(* IEC 61131-3 sources: volt/packages/volt-lsp-iec/libraries/StringUtils/3.5.18.0, 27 files *)

(* ---- CHARTOUPPER.pou ---- *)
FUNCTION CHARTOUPPER : BYTE
VAR_INPUT
	BYCHAR : BYTE;
END_VAR
(* ASCII only: a..z become A..Z, every other byte is itself *)
IF BYCHAR >= 16#61 AND BYCHAR <= 16#7A THEN
	CHARTOUPPER := BYCHAR - 16#20;
ELSE
	CHARTOUPPER := BYCHAR;
END_IF
END_FUNCTION

(* ---- HELPISSAMEIGNORECASE.pou ---- *)
FUNCTION HELPISSAMEIGNORECASE : BOOL
VAR_INPUT
	BY1 : BYTE;
	BY2 : BYTE;
END_VAR
HELPISSAMEIGNORECASE := CHARTOUPPER(BY1) = CHARTOUPPER(BY2);
END_FUNCTION

(* ---- HELPSTRCMPENDA.pou ---- *)
FUNCTION HELPSTRCMPENDA : BOOL
VAR_INPUT
	PCOMPLETETEXT : CharBufferPtr;
	PSUBTEXT : CharBufferPtr;
	XIGNORECASE : BOOL;
END_VAR
VAR
	i : DINT;
	n : DINT;
	m : DINT;
END_VAR
(* does PCOMPLETETEXT end with PSUBTEXT (case folded when XIGNORECASE) *)
IF PCOMPLETETEXT = 0 OR PSUBTEXT = 0 THEN
	RETURN;
END_IF
n := STRLENA(PCOMPLETETEXT);
m := STRLENA(PSUBTEXT);
IF m > n THEN
	RETURN;
END_IF
FOR i := 0 TO m - 1 DO
	IF XIGNORECASE THEN
		IF NOT HELPISSAMEIGNORECASE(PCOMPLETETEXT[n - m + i], PSUBTEXT[i]) THEN
			RETURN;
		END_IF
	ELSIF PCOMPLETETEXT[n - m + i] <> PSUBTEXT[i] THEN
		RETURN;
	END_IF
END_FOR
HELPSTRCMPENDA := TRUE;
END_FUNCTION

(* ---- HELPSTRCMPSTARTA.pou ---- *)
FUNCTION HELPSTRCMPSTARTA : BOOL
VAR_INPUT
	PCOMPLETETEXT : CharBufferPtr;
	PSUBTEXT : CharBufferPtr;
	XIGNORECASE : BOOL;
END_VAR
VAR
	i : DINT;
END_VAR
(* does PCOMPLETETEXT begin with PSUBTEXT — every byte of it, in order (case folded when XIGNORECASE) *)
IF PCOMPLETETEXT = 0 OR PSUBTEXT = 0 THEN
	RETURN;
END_IF
WHILE PSUBTEXT[i] <> 0 DO
	IF PCOMPLETETEXT[i] = 0 THEN
		RETURN;
	END_IF
	IF XIGNORECASE THEN
		IF NOT HELPISSAMEIGNORECASE(PCOMPLETETEXT[i], PSUBTEXT[i]) THEN
			RETURN;
		END_IF
	ELSIF PCOMPLETETEXT[i] <> PSUBTEXT[i] THEN
		RETURN;
	END_IF
	i := i + 1;
END_WHILE
HELPSTRCMPSTARTA := TRUE;
END_FUNCTION

(* ---- ISSPACECHARACTER.pou ---- *)
FUNCTION ISSPACECHARACTER : BOOL
VAR_INPUT
	WCHARACTER : WORD;
END_VAR
(* a space, one of the control characters TAB, LF, VT, FF, CR, or the no-break space 16#A0 (recorded: lib_stu_chars).
   ponytail: the other Unicode spaces (16#2000.., 16#3000) are unasked — a fixture decides them *)
ISSPACECHARACTER := WCHARACTER = 16#20 OR (WCHARACTER >= 16#09 AND WCHARACTER <= 16#0D) OR WCHARACTER = 16#A0;
END_FUNCTION

(* ---- STRCASECMPA.pou ---- *)
FUNCTION STRCASECMPA : INT
VAR_INPUT
	PBYTE1 : POINTER TO BYTE;
	PBYTE2 : POINTER TO BYTE;
END_VAR
VAR
	i : DINT;
END_VAR
(* ignoring case (ASCII), how the first bytes that differ order: -1 when PBYTE1's is lower, 1 when higher, 0 when the
   strings are equal — the sign only (recorded: lib_stu_compare) *)
IF PBYTE1 = 0 OR PBYTE2 = 0 THEN
	RETURN;
END_IF
WHILE PBYTE1[i] <> 0 AND_THEN CHARTOUPPER(PBYTE1[i]) = CHARTOUPPER(PBYTE2[i]) DO
	i := i + 1;
END_WHILE
IF CHARTOUPPER(PBYTE1[i]) < CHARTOUPPER(PBYTE2[i]) THEN
	STRCASECMPA := -1;
ELSIF CHARTOUPPER(PBYTE1[i]) > CHARTOUPPER(PBYTE2[i]) THEN
	STRCASECMPA := 1;
END_IF
END_FUNCTION

(* ---- STRCASECMPENDA.pou ---- *)
FUNCTION STRCASECMPENDA : INT
VAR_INPUT
	PSTRING : CharBufferPtr;
	PSUFFIX : CharBufferPtr;
END_VAR
(* 0 when PSTRING ends with PSUFFIX, ignoring case — the answer a compare gives for equal — and -1 when it does not *)
IF HELPSTRCMPENDA(PSTRING, PSUFFIX, TRUE) THEN
	STRCASECMPENDA := 0;
ELSE
	STRCASECMPENDA := -1;
END_IF
END_FUNCTION

(* ---- STRCASECMPSTARTA.pou ---- *)
FUNCTION STRCASECMPSTARTA : INT
VAR_INPUT
	PSTRING : CharBufferPtr;
	PPREFIX : CharBufferPtr;
END_VAR
(* 0 when PSTRING begins with PPREFIX, ignoring case — the answer a compare gives for equal — and -1 when it does not *)
IF HELPSTRCMPSTARTA(PSTRING, PPREFIX, TRUE) THEN
	STRCASECMPSTARTA := 0;
ELSE
	STRCASECMPSTARTA := -1;
END_IF
END_FUNCTION

(* ---- STRCASECMPW.pou ---- *)
FUNCTION STRCASECMPW : INT
VAR_INPUT
	PWD1 : POINTER TO WORD;
	PWD2 : POINTER TO WORD;
END_VAR
VAR
	i : DINT;
END_VAR
(* ignoring case (ASCII), how the first words that differ order: -1 when PWD1's is lower, 1 when higher, 0 when the
   strings are equal — the sign only (recorded: lib_stu_compare) *)
IF PWD1 = 0 OR PWD2 = 0 THEN
	RETURN;
END_IF
WHILE PWD1[i] <> 0 AND_THEN WCHARTOUPPER(PWD1[i]) = WCHARTOUPPER(PWD2[i]) DO
	i := i + 1;
END_WHILE
IF WCHARTOUPPER(PWD1[i]) < WCHARTOUPPER(PWD2[i]) THEN
	STRCASECMPW := -1;
ELSIF WCHARTOUPPER(PWD1[i]) > WCHARTOUPPER(PWD2[i]) THEN
	STRCASECMPW := 1;
END_IF
END_FUNCTION

(* ---- STRCASEFINDA.pou ---- *)
FUNCTION STRCASEFINDA : INT
VAR_INPUT
	PST1 : POINTER TO STRING(255);
	PST2 : POINTER TO STRING(255);
	UISEARCHSTART : UINT;
END_VAR
VAR
	i : DINT;
	j : DINT;
	n1 : DINT;
	n2 : DINT;
END_VAR
(* where PST2 first occurs in PST1, ignoring case (ASCII), searching from UISEARCHSTART (counted from 1; 0 counts as 1)
   — the position counted from 1, or 0 when it does not occur. An empty PST2 occurs nowhere. *)
IF PST1 = 0 OR PST2 = 0 THEN
	RETURN;
END_IF
WHILE PST1^[n1] <> 0 DO
	n1 := n1 + 1;
END_WHILE
WHILE PST2^[n2] <> 0 DO
	n2 := n2 + 1;
END_WHILE
IF n2 = 0 THEN
	RETURN;
END_IF
FOR i := UINT_TO_DINT(MAX(UISEARCHSTART, 1)) - 1 TO n1 - n2 DO
	j := 0;
	WHILE j < n2 AND_THEN CHARTOUPPER(PST1^[i + j]) = CHARTOUPPER(PST2^[j]) DO
		j := j + 1;
	END_WHILE
	IF j = n2 THEN
		STRCASEFINDA := DINT_TO_INT(i + 1);
		RETURN;
	END_IF
END_FOR
END_FUNCTION

(* ---- STRCASEFINDW.pou ---- *)
FUNCTION STRCASEFINDW : INT
VAR_INPUT
	PST1 : POINTER TO WSTRING(255);
	PST2 : POINTER TO WSTRING(255);
	UISEARCHSTART : UINT;
END_VAR
VAR
	i : DINT;
	j : DINT;
	n1 : DINT;
	n2 : DINT;
END_VAR
(* where PST2 first occurs in PST1, ignoring case (ASCII), searching from UISEARCHSTART (counted from 1; 0 counts as 1)
   — the position counted from 1, or 0 when it does not occur. An empty PST2 occurs nowhere. *)
IF PST1 = 0 OR PST2 = 0 THEN
	RETURN;
END_IF
WHILE PST1^[n1] <> 0 DO
	n1 := n1 + 1;
END_WHILE
WHILE PST2^[n2] <> 0 DO
	n2 := n2 + 1;
END_WHILE
IF n2 = 0 THEN
	RETURN;
END_IF
FOR i := UINT_TO_DINT(MAX(UISEARCHSTART, 1)) - 1 TO n1 - n2 DO
	j := 0;
	WHILE j < n2 AND_THEN WCHARTOUPPER(PST1^[i + j]) = WCHARTOUPPER(PST2^[j]) DO
		j := j + 1;
	END_WHILE
	IF j = n2 THEN
		STRCASEFINDW := DINT_TO_INT(i + 1);
		RETURN;
	END_IF
END_FOR
END_FUNCTION

(* ---- STRCMPA.pou ---- *)
FUNCTION STRCMPA : INT
VAR_INPUT
	PBY1 : POINTER TO BYTE;
	PBY2 : POINTER TO BYTE;
END_VAR
VAR
	i : DINT;
END_VAR
(* how the first bytes that differ order: -1 when PBY1's is lower, 1 when higher, 0 when the
   strings are equal — the sign only (recorded: lib_stu_compare) *)
IF PBY1 = 0 OR PBY2 = 0 THEN
	RETURN;
END_IF
WHILE PBY1[i] <> 0 AND_THEN PBY1[i] = PBY2[i] DO
	i := i + 1;
END_WHILE
IF PBY1[i] < PBY2[i] THEN
	STRCMPA := -1;
ELSIF PBY1[i] > PBY2[i] THEN
	STRCMPA := 1;
END_IF
END_FUNCTION

(* ---- STRCMPENDA.pou ---- *)
FUNCTION STRCMPENDA : INT
VAR_INPUT
	PSTRING : CharBufferPtr;
	PSUFFIX : CharBufferPtr;
END_VAR
(* 0 when PSTRING ends with PSUFFIX — the answer a compare gives for equal — and -1 when it does not *)
IF HELPSTRCMPENDA(PSTRING, PSUFFIX, FALSE) THEN
	STRCMPENDA := 0;
ELSE
	STRCMPENDA := -1;
END_IF
END_FUNCTION

(* ---- STRCMPSTARTA.pou ---- *)
FUNCTION STRCMPSTARTA : INT
VAR_INPUT
	PSTRING : CharBufferPtr;
	PPREFIX : CharBufferPtr;
END_VAR
(* 0 when PSTRING begins with PPREFIX — the answer a compare gives for equal — and -1 when it does not *)
IF HELPSTRCMPSTARTA(PSTRING, PPREFIX, FALSE) THEN
	STRCMPSTARTA := 0;
ELSE
	STRCMPSTARTA := -1;
END_IF
END_FUNCTION

(* ---- STRCMPW.pou ---- *)
FUNCTION STRCMPW : INT
VAR_INPUT
	PWD1 : POINTER TO WORD;
	PWD2 : POINTER TO WORD;
END_VAR
VAR
	i : DINT;
END_VAR
(* how the first words that differ order: -1 when PWD1's is lower, 1 when higher, 0 when the
   strings are equal — the sign only (recorded: lib_stu_compare) *)
IF PWD1 = 0 OR PWD2 = 0 THEN
	RETURN;
END_IF
WHILE PWD1[i] <> 0 AND_THEN PWD1[i] = PWD2[i] DO
	i := i + 1;
END_WHILE
IF PWD1[i] < PWD2[i] THEN
	STRCMPW := -1;
ELSIF PWD1[i] > PWD2[i] THEN
	STRCMPW := 1;
END_IF
END_FUNCTION

(* ---- STRCONCATA.pou ---- *)
FUNCTION STRCONCATA : BOOL
VAR_INPUT
	PSTFROM : CharBufferPtr;
	PSTTO : CharBufferPtr;
	IBUFFERSIZE : INT;
END_VAR
VAR
	i : DINT;
	nTo : DINT;
	nFrom : DINT;
END_VAR
(* PSTFROM appended to PSTTO. The result and its terminator must fit the IBUFFERSIZE bytes of PSTTO's buffer, or
   nothing is written and the answer is FALSE *)
IF PSTFROM = 0 OR PSTTO = 0 THEN
	RETURN;
END_IF
nTo := STRLENA(PSTTO);
nFrom := STRLENA(PSTFROM);
IF nTo + nFrom + 1 > IBUFFERSIZE THEN
	RETURN;
END_IF
FOR i := 0 TO nFrom - 1 DO
	PSTTO[nTo + i] := PSTFROM[i];
END_FOR
PSTTO[nTo + nFrom] := 0;
STRCONCATA := TRUE;
END_FUNCTION

(* ---- STRCPYA.pou ---- *)
FUNCTION STRCPYA : DINT
VAR_INPUT
	PBUFFER : CharBufferPtr;
	IBUFFERSIZE : DINT;
	PSTR : CharBufferPtr;
END_VAR
VAR
	i : DINT;
END_VAR
(* PSTR into the buffer, cut at the IBUFFERSIZE - 1 bytes the buffer holds before its terminator; the answer is how
   many bytes were WRITTEN, the terminator included (recorded: lib_stu_copy — 'hello' is 6, cut at 4 is 4, a buffer
   of 1 is 1) *)
IF PBUFFER = 0 OR PSTR = 0 OR IBUFFERSIZE <= 0 THEN
	RETURN;
END_IF
WHILE i < IBUFFERSIZE - 1 AND_THEN PSTR[i] <> 0 DO
	PBUFFER[i] := PSTR[i];
	i := i + 1;
END_WHILE
PBUFFER[i] := 0;
STRCPYA := i + 1;
END_FUNCTION

(* ---- STRFINDA.pou ---- *)
FUNCTION STRFINDA : INT
VAR_INPUT
	PST1 : POINTER TO STRING(255);
	PST2 : POINTER TO STRING(255);
	UISEARCHSTART : UINT;
END_VAR
VAR
	i : DINT;
	j : DINT;
	n1 : DINT;
	n2 : DINT;
END_VAR
(* where PST2 first occurs in PST1 searching from UISEARCHSTART (counted from 1; 0 counts as 1)
   — the position counted from 1, or 0 when it does not occur. An empty PST2 occurs nowhere. *)
IF PST1 = 0 OR PST2 = 0 THEN
	RETURN;
END_IF
WHILE PST1^[n1] <> 0 DO
	n1 := n1 + 1;
END_WHILE
WHILE PST2^[n2] <> 0 DO
	n2 := n2 + 1;
END_WHILE
IF n2 = 0 THEN
	RETURN;
END_IF
FOR i := UINT_TO_DINT(MAX(UISEARCHSTART, 1)) - 1 TO n1 - n2 DO
	j := 0;
	WHILE j < n2 AND_THEN PST1^[i + j] = PST2^[j] DO
		j := j + 1;
	END_WHILE
	IF j = n2 THEN
		STRFINDA := DINT_TO_INT(i + 1);
		RETURN;
	END_IF
END_FOR
END_FUNCTION

(* ---- STRFINDW.pou ---- *)
FUNCTION STRFINDW : INT
VAR_INPUT
	PST1 : POINTER TO WSTRING(255);
	PST2 : POINTER TO WSTRING(255);
	UISEARCHSTART : UINT;
END_VAR
VAR
	i : DINT;
	j : DINT;
	n1 : DINT;
	n2 : DINT;
END_VAR
(* where PST2 first occurs in PST1 searching from UISEARCHSTART (counted from 1; 0 counts as 1)
   — the position counted from 1, or 0 when it does not occur. An empty PST2 occurs nowhere. *)
IF PST1 = 0 OR PST2 = 0 THEN
	RETURN;
END_IF
WHILE PST1^[n1] <> 0 DO
	n1 := n1 + 1;
END_WHILE
WHILE PST2^[n2] <> 0 DO
	n2 := n2 + 1;
END_WHILE
IF n2 = 0 THEN
	RETURN;
END_IF
FOR i := UINT_TO_DINT(MAX(UISEARCHSTART, 1)) - 1 TO n1 - n2 DO
	j := 0;
	WHILE j < n2 AND_THEN PST1^[i + j] = PST2^[j] DO
		j := j + 1;
	END_WHILE
	IF j = n2 THEN
		STRFINDW := DINT_TO_INT(i + 1);
		RETURN;
	END_IF
END_FOR
END_FUNCTION

(* ---- STRISNULLOREMPTYA.pou ---- *)
FUNCTION STRISNULLOREMPTYA : BOOL
VAR_INPUT
	PSTDATA : CharBufferPtr;
END_VAR
IF PSTDATA = 0 THEN
	STRISNULLOREMPTYA := TRUE;
ELSE
	STRISNULLOREMPTYA := PSTDATA^ = 0;
END_IF
END_FUNCTION

(* ---- STRLENA.pou ---- *)
FUNCTION STRLENA : DINT
VAR_INPUT
	PSTDATA : CharBufferPtr;
END_VAR
(* the bytes before the terminator; a null pointer has none *)
IF PSTDATA = 0 THEN
	RETURN;
END_IF
WHILE PSTDATA[STRLENA] <> 0 DO
	STRLENA := STRLENA + 1;
END_WHILE
END_FUNCTION

(* ---- STRMIDA.pou ---- *)
FUNCTION STRMIDA
VAR_INPUT
	PST : POINTER TO BYTE;
	UIINPUTBUFFERSIZE : UINT;
	ILENGTH : INT;
	IPOSITION : INT;
	PSTRESULT : POINTER TO BYTE;
	UIRESULTBUFFERSIZE : UINT;
END_VAR
VAR
	i : DINT;
	n : DINT;
END_VAR
(* ILENGTH characters of PST from IPOSITION (counted from 1) into PSTRESULT, cut at the UIRESULTBUFFERSIZE - 1 bytes
   it holds before its terminator — MID over byte buffers. PSTRESULT may be PST itself: each byte is read before it
   is written over. A position before the first character or past the last leaves PSTRESULT as it was (recorded:
   lib_stu_mid); a length of 0 empties it. ponytail: a position just past the end (length + 1) is unasked *)
IF PST = 0 OR PSTRESULT = 0 OR UIRESULTBUFFERSIZE = 0 THEN
	RETURN;
END_IF
n := STRLENA(PST);
IF IPOSITION < 1 OR IPOSITION > n THEN
	RETURN;
END_IF
n := n - (IPOSITION - 1);
n := MIN(n, ILENGTH, UINT_TO_DINT(UIRESULTBUFFERSIZE) - 1);
FOR i := 0 TO n - 1 DO
	PSTRESULT[i] := PST[IPOSITION - 1 + i];
END_FOR
PSTRESULT[MAX(n, 0)] := 0;
END_FUNCTION

(* ---- STRPADLEFTA.pou ---- *)
FUNCTION STRPADLEFTA : BOOL
VAR_INPUT
	BYPADCHAR : BYTE;
	PSTFROM : CharBufferPtr;
	PSTTO : CharBufferPtr;
	DIBUFFERSIZE : DINT;
END_VAR
VAR
	i : DINT;
	n : DINT;
	pad : DINT;
END_VAR
(* PSTFROM, filled up on the LEFT with BYPADCHAR to DIBUFFERSIZE characters, into PSTTO (recorded: lib_stu_pad —
   'abc' to 6 is '***abc'). A source that is already longer does not fit: nothing is written and the answer is FALSE *)
IF PSTFROM = 0 OR PSTTO = 0 THEN
	RETURN;
END_IF
n := STRLENA(PSTFROM);
pad := DIBUFFERSIZE - n;
IF pad < 0 THEN
	RETURN;
END_IF
FOR i := 0 TO pad - 1 DO
	PSTTO[i] := BYPADCHAR;
END_FOR
FOR i := 0 TO n - 1 DO
	PSTTO[pad + i] := PSTFROM[i];
END_FOR
PSTTO[pad + n] := 0;
STRPADLEFTA := TRUE;
END_FUNCTION

(* ---- STRPADRIGHTA.pou ---- *)
FUNCTION STRPADRIGHTA : BOOL
VAR_INPUT
	BYPADCHAR : BYTE;
	PSTFROM : CharBufferPtr;
	PSTTO : CharBufferPtr;
	DIBUFFERSIZE : DINT;
END_VAR
VAR
	i : DINT;
	n : DINT;
END_VAR
(* PSTFROM, filled up on the RIGHT with BYPADCHAR to DIBUFFERSIZE characters, into PSTTO (recorded: lib_stu_pad —
   'abc' to 6 is 'abc...'). A source that is already longer does not fit: nothing is written and the answer is FALSE *)
IF PSTFROM = 0 OR PSTTO = 0 THEN
	RETURN;
END_IF
n := STRLENA(PSTFROM);
IF n > DIBUFFERSIZE THEN
	RETURN;
END_IF
FOR i := 0 TO n - 1 DO
	PSTTO[i] := PSTFROM[i];
END_FOR
FOR i := n TO DIBUFFERSIZE - 1 DO
	PSTTO[i] := BYPADCHAR;
END_FOR
PSTTO[DIBUFFERSIZE] := 0;
STRPADRIGHTA := TRUE;
END_FUNCTION

(* ---- STRREPLACEA.pou ---- *)
FUNCTION STRREPLACEA
VAR_INPUT
	PSTINPUT : POINTER TO STRING(255);
	UIINPUTBUFFERSIZE : UINT;
	PSTREPLACEWITH : POINTER TO STRING(255);
	ILENGTHINPUT : INT;
	ILENGTHTOREPLACE : INT;
	ILENGTHTOREPLACEWITH : INT;
	IPOSITION : INT;
END_VAR
VAR
	buf : ARRAY[0..255] OF BYTE;
	i : DINT;
	n : DINT;
	p : DINT;
	cnt : DINT;
	src : DINT;
	dst : DINT;
	cap : DINT;
END_VAR
(* NOT REPLACE — a raw in-place move over the input's BUFFER, as CODESYS answers it (recorded: lib_stu_replace,
   lib_stu_replace_past_len). With p = IPOSITION - 1:
   1. the bytes from p + ILENGTHTOREPLACE up to ILENGTHINPUT, its terminator included, move to p + ILENGTHTOREPLACEWITH
      — nothing moves when ILENGTHINPUT does not reach past them, so ILENGTHINPUT is the input's LENGTH and a wrong
      one leaves the tail where it was ('abcdef', 1 at 4, length 1 → 'abcXYZ'); one past the length moves the bytes
      behind the terminator too ('abcdefghijkl' := 'abc', 3 for 1 at 2, length 12 → 'aXYZghijkl');
   2. the WHOLE of PSTREPLACEWITH is copied over p — its length is not ILENGTHTOREPLACEWITH ('Device.App', 1 for 1 at
      7 → 'DeviceXYZp') — at any position inside the buffer, behind the terminator too.
   Both are cut at UIINPUTBUFFERSIZE - 1, with a terminator there when anything moved. The buffer is read and written
   back whole, up to that size, so what lies behind the terminator is moved as CODESYS moves it in place.
   ponytail: a buffer larger than 255 is not modelled
   A UIINPUTBUFFERSIZE larger than the caller's string is not modelled either: CODESYS reads and writes the bytes behind
   the variable (buf[cap] := 0 lands in the neighbour), the model faults at run time on the first unit past the string's
   capacity. niche: accepted loss (0 occurrences in the corpora: the one caller, pro2193 ParseInstanceName, passes 80 for
   a STRING(80)) *)
IF PSTINPUT = 0 OR PSTREPLACEWITH = 0 OR IPOSITION < 1 THEN
	RETURN;
END_IF
cap := MIN(UINT_TO_DINT(UIINPUTBUFFERSIZE) - 1, 255);
FOR i := 0 TO cap DO
	buf[i] := PSTINPUT^[i];
END_FOR
p := IPOSITION - 1;
cnt := ILENGTHINPUT - p - ILENGTHTOREPLACE + 1;
src := p + ILENGTHTOREPLACE;
dst := p + ILENGTHTOREPLACEWITH;
IF cnt > 0 THEN
	cnt := MIN(cnt, MIN(cap - dst, cap - src));
	IF dst > src THEN
		FOR i := cnt - 1 TO 0 BY -1 DO
			buf[dst + i] := buf[src + i];
		END_FOR
	ELSE
		FOR i := 0 TO cnt - 1 DO
			buf[dst + i] := buf[src + i];
		END_FOR
	END_IF
	buf[cap] := 0;
END_IF
i := 0;
WHILE PSTREPLACEWITH^[i] <> 0 AND p + i < cap DO
	buf[p + i] := PSTREPLACEWITH^[i];
	i := i + 1;
END_WHILE
FOR i := 0 TO cap DO
	PSTINPUT^[i] := buf[i];
END_FOR
END_FUNCTION

(* ---- STRTRIMA.pou ---- *)
FUNCTION STRTRIMA
VAR_INPUT
	PSTRING : POINTER TO BYTE;
END_VAR
VAR
	i : DINT;
	first : DINT;
	last : DINT;
END_VAR
(* PSTRING without its leading and trailing spaces (ISSPACECHARACTER), in place *)
IF PSTRING = 0 THEN
	RETURN;
END_IF
last := STRLENA(PSTRING) - 1;
WHILE first <= last AND_THEN ISSPACECHARACTER(PSTRING[first]) DO
	first := first + 1;
END_WHILE
WHILE last >= first AND_THEN ISSPACECHARACTER(PSTRING[last]) DO
	last := last - 1;
END_WHILE
FOR i := 0 TO last - first DO
	PSTRING[i] := PSTRING[first + i];
END_FOR
PSTRING[MAX(last - first + 1, 0)] := 0;
END_FUNCTION

(* ---- WCHARTOUPPER.pou ---- *)
FUNCTION WCHARTOUPPER : WORD
VAR_INPUT
	WDCHAR : WORD;
END_VAR
(* ASCII only, as CharToUpper: a..z become A..Z, every other unit is itself *)
IF WDCHAR >= 16#61 AND WDCHAR <= 16#7A THEN
	WCHARTOUPPER := WDCHAR - 16#20;
ELSE
	WCHARTOUPPER := WDCHAR;
END_IF
END_FUNCTION
